# EPICS substitutions: apps/caenHvApp/Db/seq/fttfthOnOff.substitutions
file "db/fttOnOff.db" {
pattern { ONOFF VAL }
    { OFF 0 }
    { ON 1 }
}
file "db/fthOnOff.db" {
pattern { ONOFF VAL }
    { OFF 0 }
    { ON 1 }
}
